(* PLC project Sin nombre, Desconocido Sin nombre 1 *)
(* stored: creationDateTime 2024-11-27T12:18:52, modificationDateTime 2024-11-27T12:35:24 *)

PROGRAM rele
  VAR
    BTN_INICIO : BOOL;
    BTN_PARO : BOOL;
    M_MOTOR : BOOL;
    MOTOR : BOOL;
  END_VAR

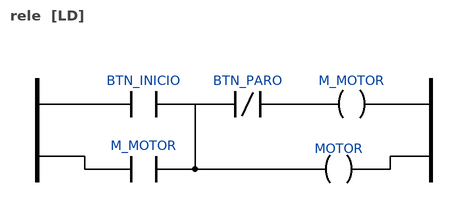
(* LD diagram, written out as Structured Text *)
M_MOTOR := (BTN_INICIO OR M_MOTOR) AND NOT BTN_PARO;
MOTOR := M_MOTOR;
END_PROGRAM

CONFIGURATION Config0
  RESOURCE Res0 ON PLC
    TASK task0(INTERVAL := T#20ms, PRIORITY := 0);
    PROGRAM instance0 WITH task0 : rele;
  END_RESOURCE
END_CONFIGURATION
